(* Schneider Machine Expert - Basic project Ochistka, file version 2.6.0.0 *)
(* ProjectInformations: Name=New project *)

HARDWARE
  Cpu 0: TM221CE40T
  ModuleExtensionObject 0: TM3DI32K
  ModuleExtensionObject 1: TM3DI32K
  ModuleExtensionObject 2: TM3DI32K
  ModuleExtensionObject 3: TM3DI32K
  ModuleExtensionObject 4: TM3DI32K
  ModuleExtensionObject 5: TM3DI32K
  ModuleExtensionObject 6: TM3DQ32TK
  EthernetConfiguration: NetworkName=M221, IpAllocationMode=FixedAddress, IpAddress=0.0.0.0, SubnetMask=0.0.0.0
  SerialLineConfiguration: Baud=Baud19200, Parity=ParityEven, DataBits=DataBits8, StopBits=StopBits1, PhysicalMedium=PhysicalMediumRs485, TransmissionMode=TransmissionModeModbusRtu, SlaveId=1, Addressing=SlaveAddressing
  MastTask: UsePeriodScanMode=false, PeriodScan=100
  FastTask: Period=255
  CpuBehavior: StartingMode=StartAsPreviousState, AutoSaveRamOnEeprom=true, WatchdogPeriod=250

SYMBOLS  (address, symbol, comment, settings)
  %M0       PUSK_SISTEM
  %M1       EMG_STOP_SHKAF
  %M2       EMG_STOP_BIG_BAG
  %M3       EMG_STOP_TRIER
  %M4       EMG_STOP
  %M5       ERR_RKF
  %M6       RUN_SIRENA
  %M7       RUN_ALARM
  %M8       DP_KONVEER_2
  %M9       BTN_LPUSK_KONVEER_2
  %M10      BTN_LSTOP_KONVEER_2
  %M11      ERR_PCH_KONVEER_2
  %M12      RUN_KONVEER_2
  %M13      RESET_ERR_PCH_KONVEER_2

POU Input_A1
  (* SectionNumber=0 *)

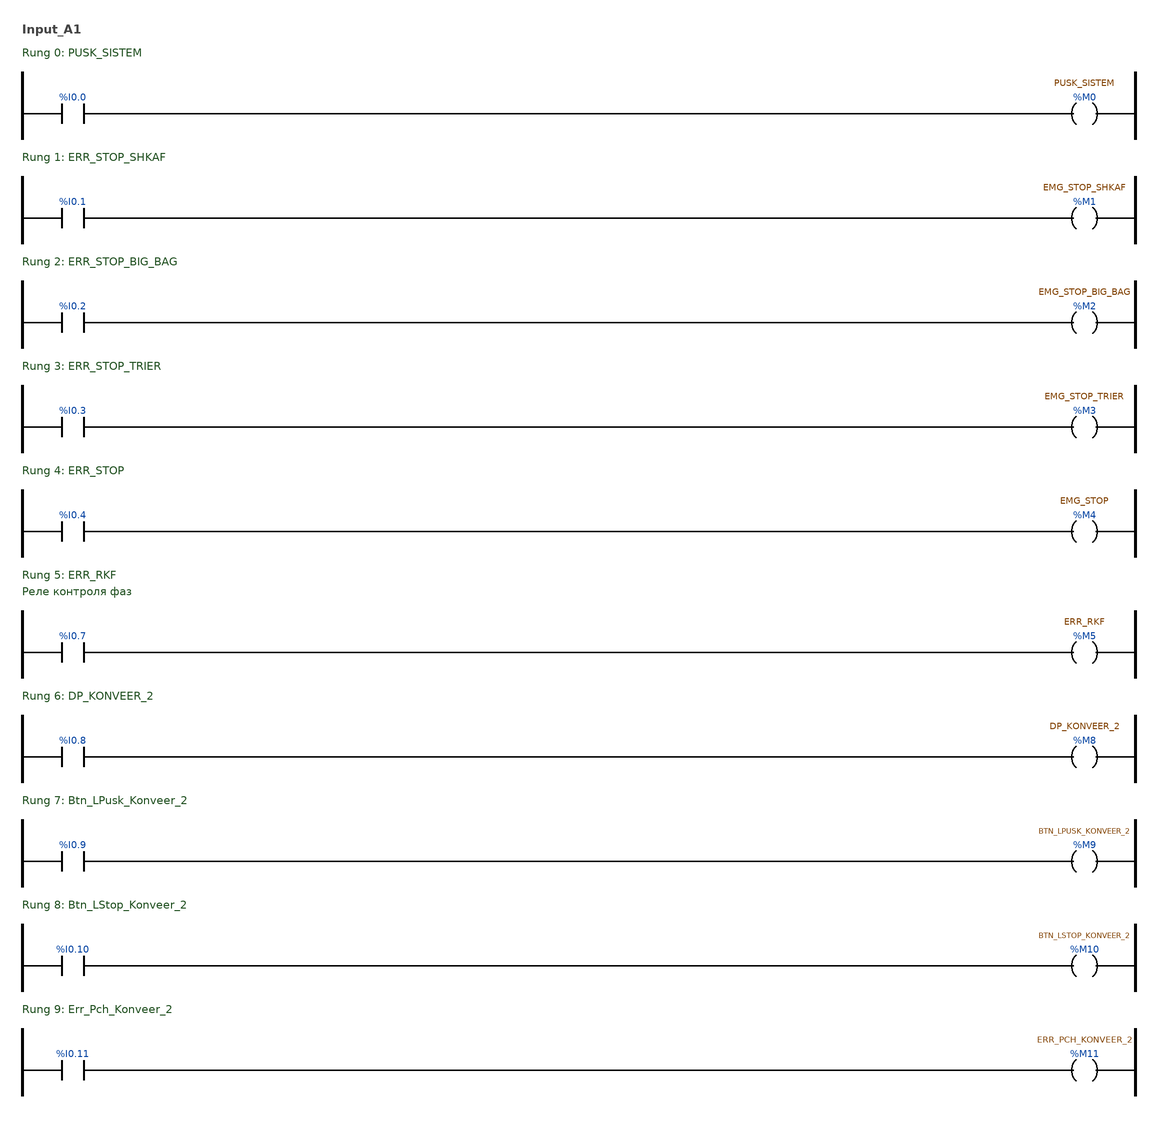

// Rung 0: PUSK_SISTEM
  LD %I0.0
  ST %M0                  (* PUSK_SISTEM *)
  // as ST:
  //   PUSK_SISTEM := %I0.0;

// Rung 1: ERR_STOP_SHKAF
  LD %I0.1
  ST %M1                  (* EMG_STOP_SHKAF *)
  // as ST:
  //   EMG_STOP_SHKAF := %I0.1;

// Rung 2: ERR_STOP_BIG_BAG
  LD %I0.2
  ST %M2                  (* EMG_STOP_BIG_BAG *)
  // as ST:
  //   EMG_STOP_BIG_BAG := %I0.2;

// Rung 3: ERR_STOP_TRIER
  LD %I0.3
  ST %M3                  (* EMG_STOP_TRIER *)
  // as ST:
  //   EMG_STOP_TRIER := %I0.3;

// Rung 4: ERR_STOP
  LD %I0.4
  ST %M4                  (* EMG_STOP *)
  // as ST:
  //   EMG_STOP := %I0.4;

// Rung 5: ERR_RKF
// Реле контроля фаз
  LD %I0.7
  ST %M5                  (* ERR_RKF *)
  // as ST:
  //   ERR_RKF := %I0.7;

// Rung 6: DP_KONVEER_2
  LD %I0.8
  ST %M8                  (* DP_KONVEER_2 *)
  // as ST:
  //   DP_KONVEER_2 := %I0.8;

// Rung 7: Btn_LPusk_Konveer_2
  LD %I0.9
  ST %M9                  (* BTN_LPUSK_KONVEER_2 *)
  // as ST:
  //   BTN_LPUSK_KONVEER_2 := %I0.9;

// Rung 8: Btn_LStop_Konveer_2
  LD %I0.10
  ST %M10                 (* BTN_LSTOP_KONVEER_2 *)
  // as ST:
  //   BTN_LSTOP_KONVEER_2 := %I0.10;

// Rung 9: Err_Pch_Konveer_2
  LD %I0.11
  ST %M11                 (* ERR_PCH_KONVEER_2 *)
  // as ST:
  //   ERR_PCH_KONVEER_2 := %I0.11;

POU Output_A1
  (* SectionNumber=0 *)

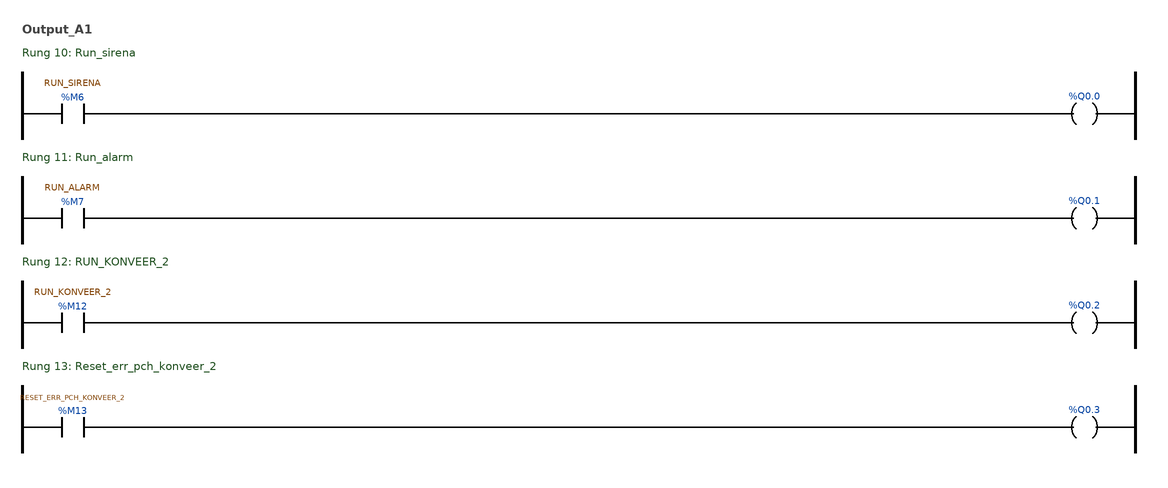

// Rung 10: Run_sirena
  LD %M6                  (* RUN_SIRENA *)
  ST %Q0.0
  // as ST:
  //   %Q0.0 := RUN_SIRENA;

// Rung 11: Run_alarm
  LD %M7                  (* RUN_ALARM *)
  ST %Q0.1
  // as ST:
  //   %Q0.1 := RUN_ALARM;

// Rung 12: RUN_KONVEER_2
  LD %M12                 (* RUN_KONVEER_2 *)
  ST %Q0.2
  // as ST:
  //   %Q0.2 := RUN_KONVEER_2;

// Rung 13: Reset_err_pch_konveer_2
  LD %M13                 (* RESET_ERR_PCH_KONVEER_2 *)
  ST %Q0.3
  // as ST:
  //   %Q0.3 := RESET_ERR_PCH_KONVEER_2;
